% RSLogix 500 project LAB2.RSS, saved by version 8.10.00.30 %
PROJECT "LAB2.2"    % processor: Bul.1763 MicroLogix 1100 Series A %

PROGRAM FILES
  LAD 2   15 rungs

DATA FILES
  O0 OUTPUT  4 elements
  I1 INPUT  6 elements
  S2 STATUS  66 elements
  B3 BINARY  1 elements
  T4 TIMER  2 elements
  C5 COUNTER  1 elements
  R6 CONTROL  1 elements
  N7 INTEGER  1 elements
  F8 FLOAT  1 elements

LADDER 2
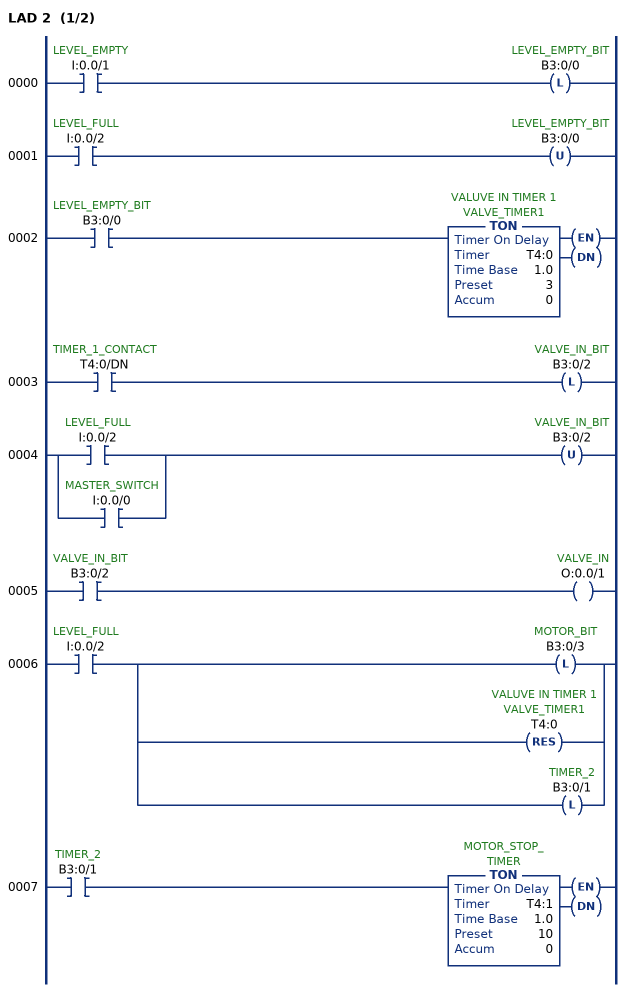
% Rung: 0 %
SOR XIC I:0.0/1 OTL B3:0/0 EOR
%   I:0.0/1  LEVEL_EMPTY %
%   B3:0/0  LEVEL_EMPTY_BIT %
% Rung: 1 %
SOR XIC I:0.0/2 OTU B3:0/0 EOR
%   I:0.0/2  LEVEL_FULL %
%   B3:0/0  LEVEL_EMPTY_BIT %
% Rung: 2 %
SOR XIC B3:0/0 TON T4:0 1.0 3 0 EOR
%   B3:0/0  LEVEL_EMPTY_BIT %
%   T4:0  VALVE_TIMER1  "VALUVE IN TIMER 1" %
% Rung: 3 %
SOR XIC T4:0/DN OTL B3:0/2 EOR
%   T4:0/DN  TIMER_1_CONTACT %
%   B3:0/2  VALVE_IN_BIT %
% Rung: 4 %
SOR BST XIC I:0.0/2 NXB XIC I:0.0/0 BND OTU B3:0/2 EOR
%   I:0.0/2  LEVEL_FULL %
%   I:0.0/0  MASTER_SWITCH %
%   B3:0/2  VALVE_IN_BIT %
% Rung: 5 %
SOR XIC B3:0/2 OTE O:0.0/1 EOR
%   B3:0/2  VALVE_IN_BIT %
%   O:0.0/1  VALVE_IN %
% Rung: 6 %
SOR XIC I:0.0/2 BST OTL B3:0/3 NXB BST RES T4:0 NXB OTL B3:0/1 BND BND EOR
%   I:0.0/2  LEVEL_FULL %
%   B3:0/3  MOTOR_BIT %
%   T4:0  VALVE_TIMER1  "VALUVE IN TIMER 1" %
%   B3:0/1  TIMER_2 %
% Rung: 7 %
SOR XIC B3:0/1 TON T4:1 1.0 10 0 EOR
%   B3:0/1  TIMER_2 %
%   T4:1  MOTOR_STOP_TIMER %

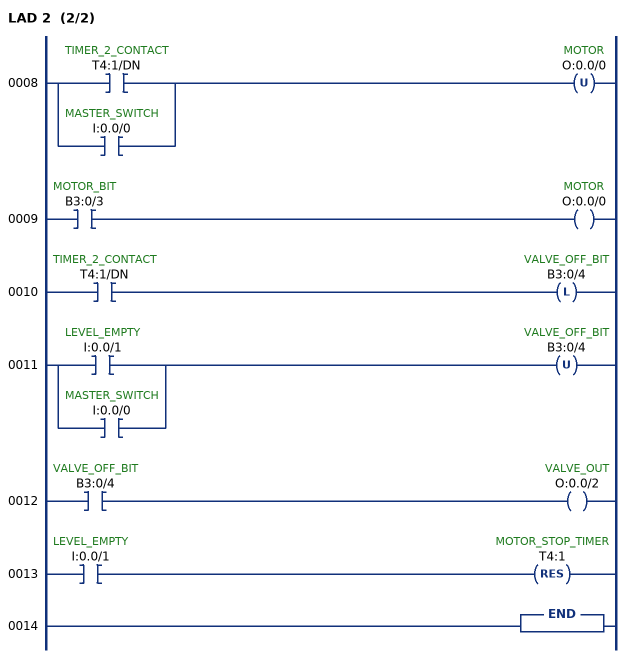
% Rung: 8 %
SOR BST XIC T4:1/DN NXB XIC I:0.0/0 BND OTU O:0.0/0 EOR
%   T4:1/DN  TIMER_2_CONTACT %
%   I:0.0/0  MASTER_SWITCH %
%   O:0.0/0  MOTOR %
% Rung: 9 %
SOR XIC B3:0/3 OTE O:0.0/0 EOR
%   B3:0/3  MOTOR_BIT %
%   O:0.0/0  MOTOR %
% Rung: 10 %
SOR XIC T4:1/DN OTL B3:0/4 EOR
%   T4:1/DN  TIMER_2_CONTACT %
%   B3:0/4  VALVE_OFF_BIT %
% Rung: 11 %
SOR BST XIC I:0.0/1 NXB XIC I:0.0/0 BND OTU B3:0/4 EOR
%   I:0.0/1  LEVEL_EMPTY %
%   I:0.0/0  MASTER_SWITCH %
%   B3:0/4  VALVE_OFF_BIT %
% Rung: 12 %
SOR XIC B3:0/4 OTE O:0.0/2 EOR
%   B3:0/4  VALVE_OFF_BIT %
%   O:0.0/2  VALVE_OUT %
% Rung: 13 %
SOR XIC I:0.0/1 RES T4:1 EOR
%   I:0.0/1  LEVEL_EMPTY %
%   T4:1  MOTOR_STOP_TIMER %
% Rung: 14 %
SOR END EOR

DATA TABLE (non-zero values as saved)
DATA T4
% .PRE .ACC %
% T4:0 % 3 0
% T4:1 % 10 0
